// TIA Portal V16 export
// export: Created 2024-09-05T17:39:09.6255784Z, ExportSetting WithDefaults, DisplayName Totally Integrated Automation Portal, DisplayVersion V16 Update 6, DisplayName TIA Portal Version Control Interface, DisplayVersion V16 Update 2, DisplayName TIA Portal Openness, DisplayVersion V16 Update 6, DisplayName STEP 7 Professional, DisplayVersion V16 Update 6, DisplayName STEP 7 Safety, DisplayVersion V16, DisplayName WinCC Advanced, DisplayVersion V16 Update 6
DATA_BLOCK "CylindersHMI"   // DB50
{ S7_Optimized_Access := 'TRUE' }
VERSION : 0.1
// stored: AutoNumber true, DBAccessibleFromOPCUA true, IsOnlyStoredInLoadMemory false, IsRetainMemResEnabled false, IsWriteProtectedInAS false, MemoryReserve 100
   VAR
      Status : Array[0.."NumberOfCylinders"] of Int;
      SelectedCylinderCylinderCommand : Int := 0;
      SelectedCylinder : Int := 0;
      SelectedCylinderStatus : Int := 0;
      SelectedCylinder_1 : Int := 0;
      SelectedCylinder_2 : Int := 0;
      SelectedCylinder_3 : Int := 0;
      SelectedCylinder_4 : Int := 0;
      SelectedCylinderStatus_1 : Int := 0;
      SelectedCylinderStatus_2 : Int := 0;
      SelectedCylinderStatus_3 : Int := 0;
      SelectedCylinderStatus_4 : Int := 0;
      DisableHMIControl : Bool := FALSE;
      CylinderInfoHMI : Int := -1;
      CylinderInfoHMIAction : Int := 0;
   END_VAR
BEGIN
   Status[0..4] := 257;
   Status[5..6] := 1;
   Status[7..8] := 257;
   Status[9..10] := 1;
   Status[11..14] := 257;
   Status[15..16] := 1;
   Status[17] := 2;
   Status[18] := 1;
   Status[19] := 0;
END_DATA_BLOCK
